FUNCTION "FC2027_ZC_FF_SEC" : Void
TITLE = FC2027_FF_SEC
{ S7_Optimized_Access := 'TRUE' }
AUTHOR : ABH
FAMILY : ZeusControl
VERSION : 1.0
//Funcion para gestion de Flip Flop secuencial.
   VAR_INPUT
      Pulso1Seg : Bool;   // Pulso de 1 segundo
   END_VAR

   VAR_TEMP
      for_i : Int;
      t_Flip_1 : Int;
      t_Flip_2 : Int;
      t_Flip_3 : Int;
      t_Flip_4 : Int;
      t_Flip_5 : Int;
      t_Flip_6 : Int;
      t_Flip_7 : Int;
      t_Flip_8 : Int;
      t_Flip_9 : Int;
      t_Flip_10 : Int;
   END_VAR


BEGIN
	(*
	ZEUS CONTROL, S.A.
	(c)Copyright (2023) All Rights Reserved
	--------------------------------------------------------------------------------------

	Software:       TIA Portal 16
	Restricciones:  PLC serie 1200/1500

	Nombre:         DISPOSITIVO FLIP FLOP SECUENCIAL
	Descripcion:    Modelo de dispositivo Flip Flop Secuencial

	Dependencias:
	    FC:         -
	    FB:         -
	    UDT:        ZC_DISP_FF_SEC
	    DB:         DB2027_DISP_FF_SEC

	Change log:

	    Version     Fecha       Tecnico a cargo     Descripcion

	    01.00.00    23.06.2022  (ABH)               Primera version
	    01.00.01    15.07.2022  (HCR)               Se aumenta la gestion de flips de 6 a 10.
	    01.00.02    28.11.2023  (ABH)               Se añade condicion de activacion del Flip Flop a que algun SP sea mayor que 0.
	    01.00.03    15.10.2025  (ABH)               Se añade orden pausa para dejar de contar.

	//=====================================================================================
	*)



	FOR #for_i := 1 TO "N_MAX_DISP_FF_SEC" DO


	    IF "DB2027_FF_SEC".FF_SEC[#for_i].Orden_Activar AND
	        ("DB2027_FF_SEC".FF_SEC[#for_i].Config_SetPointTiempoFlip1 > 0
	        OR"DB2027_FF_SEC".FF_SEC[#for_i].Config_SetPointTiempoFlip2 > 0
	        OR"DB2027_FF_SEC".FF_SEC[#for_i].Config_SetPointTiempoFlip3 > 0
	        OR"DB2027_FF_SEC".FF_SEC[#for_i].Config_SetPointTiempoFlip4 > 0
	        OR"DB2027_FF_SEC".FF_SEC[#for_i].Config_SetPointTiempoFlip5 > 0
	        OR"DB2027_FF_SEC".FF_SEC[#for_i].Config_SetPointTiempoFlip6 > 0
	        OR"DB2027_FF_SEC".FF_SEC[#for_i].Config_SetPointTiempoFlip7 > 0
	        OR"DB2027_FF_SEC".FF_SEC[#for_i].Config_SetPointTiempoFlip8 > 0
	        OR"DB2027_FF_SEC".FF_SEC[#for_i].Config_SetPointTiempoFlip9 > 0
	        OR"DB2027_FF_SEC".FF_SEC[#for_i].Config_SetPointTiempoFlip10 > 0
	        OR"DB2027_FF_SEC".FF_SEC[#for_i].Config_SetPointTiempoFlop > 0)
	    THEN



	        REGION ARRANQUE_ACTIVACION_FLOP

	            //  EN EL ARRANQUE SE ACTIVA FLOP
	            IF "DB2027_FF_SEC".FF_SEC[#for_i].Aux_Flanco = FALSE THEN
	                "DB2027_FF_SEC".FF_SEC[#for_i].Aux_FlopActivo := TRUE;
	                "DB2027_FF_SEC".FF_SEC[#for_i].Aux_FlipActivo := FALSE;
	                "DB2027_FF_SEC".FF_SEC[#for_i].Aux_Flanco := TRUE;
	            END_IF;

	        END_REGION


	        REGION CALCULO_TIEMPOS_FLIP

	            //  CALCULO DE ACTIVACIONES SECUENCIALES
	            #t_Flip_1 := "DB2027_FF_SEC".FF_SEC[#for_i].Config_SetPointTiempoFlip1;
	            #t_Flip_2 := #t_Flip_1 + "DB2027_FF_SEC".FF_SEC[#for_i].Config_SetPointTiempoFlip2;
	            #t_Flip_3 := #t_Flip_2 + "DB2027_FF_SEC".FF_SEC[#for_i].Config_SetPointTiempoFlip3;
	            #t_Flip_4 := #t_Flip_3 + "DB2027_FF_SEC".FF_SEC[#for_i].Config_SetPointTiempoFlip4;
	            #t_Flip_5 := #t_Flip_4 + "DB2027_FF_SEC".FF_SEC[#for_i].Config_SetPointTiempoFlip5;
	            #t_Flip_6 := #t_Flip_5 + "DB2027_FF_SEC".FF_SEC[#for_i].Config_SetPointTiempoFlip6;
	            #t_Flip_7 := #t_Flip_6 + "DB2027_FF_SEC".FF_SEC[#for_i].Config_SetPointTiempoFlip7;
	            #t_Flip_8 := #t_Flip_7 + "DB2027_FF_SEC".FF_SEC[#for_i].Config_SetPointTiempoFlip8;
	            #t_Flip_9 := #t_Flip_8 + "DB2027_FF_SEC".FF_SEC[#for_i].Config_SetPointTiempoFlip9;
	            #t_Flip_10 := #t_Flip_9 + "DB2027_FF_SEC".FF_SEC[#for_i].Config_SetPointTiempoFlip10;

	            //  CALCULO DE TIEMPO FLIP TOTAL
	            "DB2027_FF_SEC".FF_SEC[#for_i].Aux_TiempoFlipTotal :=
	            "DB2027_FF_SEC".FF_SEC[#for_i].Config_SetPointTiempoFlip1 +
	            "DB2027_FF_SEC".FF_SEC[#for_i].Config_SetPointTiempoFlip2 +
	            "DB2027_FF_SEC".FF_SEC[#for_i].Config_SetPointTiempoFlip3 +
	            "DB2027_FF_SEC".FF_SEC[#for_i].Config_SetPointTiempoFlip4 +
	            "DB2027_FF_SEC".FF_SEC[#for_i].Config_SetPointTiempoFlip5 +
	            "DB2027_FF_SEC".FF_SEC[#for_i].Config_SetPointTiempoFlip6 +
	            "DB2027_FF_SEC".FF_SEC[#for_i].Config_SetPointTiempoFlip7 +
	            "DB2027_FF_SEC".FF_SEC[#for_i].Config_SetPointTiempoFlip8 +
	            "DB2027_FF_SEC".FF_SEC[#for_i].Config_SetPointTiempoFlip9 +
	            "DB2027_FF_SEC".FF_SEC[#for_i].Config_SetPointTiempoFlip10;

	        END_REGION


	        REGION ACTIVACION_FLIP_FLOP

	            //  GESTION FLIP
	            IF "DB2027_FF_SEC".FF_SEC[#for_i].Aux_TiempoFlip >= "DB2027_FF_SEC".FF_SEC[#for_i].Aux_TiempoFlipTotal THEN

	                "DB2027_FF_SEC".FF_SEC[#for_i].Aux_TiempoFlip := 0;
	                "DB2027_FF_SEC".FF_SEC[#for_i].Aux_FlipActivo := FALSE;
	                "DB2027_FF_SEC".FF_SEC[#for_i].Aux_FlopActivo := TRUE;

	            END_IF;

	            //  GESTION FLOP
	            IF "DB2027_FF_SEC".FF_SEC[#for_i].Aux_TiempoFlop >= "DB2027_FF_SEC".FF_SEC[#for_i].Config_SetPointTiempoFlop THEN

	                "DB2027_FF_SEC".FF_SEC[#for_i].Aux_TiempoFlop := 0;
	                "DB2027_FF_SEC".FF_SEC[#for_i].Aux_FlipActivo := TRUE;
	                "DB2027_FF_SEC".FF_SEC[#for_i].Aux_FlopActivo := FALSE;

	            END_IF;

	        END_REGION


	        REGION CONTAJE_TIEMPOS_FLIP_FLOP

	            IF #Pulso1Seg AND NOT "DB2027_FF_SEC".FF_SEC[#for_i].Orden_Pausa THEN

	                //  CUENTA FLIP
	                IF "DB2027_FF_SEC".FF_SEC[#for_i].Aux_FlipActivo THEN
	                    "DB2027_FF_SEC".FF_SEC[#for_i].Aux_TiempoFlip += + 1;
	                END_IF;

	                //  CUENTA FLOP
	                IF "DB2027_FF_SEC".FF_SEC[#for_i].Aux_FlopActivo THEN
	                    "DB2027_FF_SEC".FF_SEC[#for_i].Aux_TiempoFlop += + 1;
	                END_IF;

	            END_IF;

	        END_REGION


	        REGION ACTIVACION_SALIDAS

	            // GESTION SALIDAS FLOP
	            IF "DB2027_FF_SEC".FF_SEC[#for_i].Aux_FlopActivo THEN

	                "DB2027_FF_SEC".FF_SEC[#for_i].Estado_SalidaFlop := TRUE;

	                "DB2027_FF_SEC".FF_SEC[#for_i].Estado_SalidaFlip1 :=
	                "DB2027_FF_SEC".FF_SEC[#for_i].Estado_SalidaFlip2 :=
	                "DB2027_FF_SEC".FF_SEC[#for_i].Estado_SalidaFlip3 :=
	                "DB2027_FF_SEC".FF_SEC[#for_i].Estado_SalidaFlip4 :=
	                "DB2027_FF_SEC".FF_SEC[#for_i].Estado_SalidaFlip5 :=
	                "DB2027_FF_SEC".FF_SEC[#for_i].Estado_SalidaFlip6 :=
	                "DB2027_FF_SEC".FF_SEC[#for_i].Estado_SalidaFlip7 :=
	                "DB2027_FF_SEC".FF_SEC[#for_i].Estado_SalidaFlip8 :=
	                "DB2027_FF_SEC".FF_SEC[#for_i].Estado_SalidaFlip9 :=
	                "DB2027_FF_SEC".FF_SEC[#for_i].Estado_SalidaFlip10 := FALSE;
	            END_IF;

	            // GESTION SALIDAS FLIP
	            IF "DB2027_FF_SEC".FF_SEC[#for_i].Aux_FlipActivo THEN

	                //  ACTIVACION FLIP 1
	                IF "DB2027_FF_SEC".FF_SEC[#for_i].Aux_TiempoFlip < #t_Flip_1 AND "DB2027_FF_SEC".FF_SEC[#for_i].Config_SetPointTiempoFlip1 <> 0 THEN
	                    "DB2027_FF_SEC".FF_SEC[#for_i].Estado_SalidaFlip1 := TRUE;
	                ELSE
	                    "DB2027_FF_SEC".FF_SEC[#for_i].Estado_SalidaFlip1 := FALSE;
	                END_IF;

	                //  ACTIVACION FLIP 2
	                IF "DB2027_FF_SEC".FF_SEC[#for_i].Aux_TiempoFlip >= #t_Flip_1 AND "DB2027_FF_SEC".FF_SEC[#for_i].Aux_TiempoFlip < #t_Flip_2 AND "DB2027_FF_SEC".FF_SEC[#for_i].Config_SetPointTiempoFlip2 <> 0 THEN
	                    "DB2027_FF_SEC".FF_SEC[#for_i].Estado_SalidaFlip2 := TRUE;
	                ELSE
	                    "DB2027_FF_SEC".FF_SEC[#for_i].Estado_SalidaFlip2 := FALSE;
	                END_IF;

	                //  ACTIVACION FLIP 3
	                IF "DB2027_FF_SEC".FF_SEC[#for_i].Aux_TiempoFlip >= #t_Flip_2 AND "DB2027_FF_SEC".FF_SEC[#for_i].Aux_TiempoFlip < #t_Flip_3 AND "DB2027_FF_SEC".FF_SEC[#for_i].Config_SetPointTiempoFlip3 <> 0 THEN
	                    "DB2027_FF_SEC".FF_SEC[#for_i].Estado_SalidaFlip3 := TRUE;
	                ELSE
	                    "DB2027_FF_SEC".FF_SEC[#for_i].Estado_SalidaFlip3 := FALSE;
	                END_IF;

	                //  ACTIVACION FLIP 4
	                IF "DB2027_FF_SEC".FF_SEC[#for_i].Aux_TiempoFlip >= #t_Flip_3 AND "DB2027_FF_SEC".FF_SEC[#for_i].Aux_TiempoFlip < #t_Flip_4 AND "DB2027_FF_SEC".FF_SEC[#for_i].Config_SetPointTiempoFlip4 <> 0 THEN
	                    "DB2027_FF_SEC".FF_SEC[#for_i].Estado_SalidaFlip4 := TRUE;
	                ELSE
	                    "DB2027_FF_SEC".FF_SEC[#for_i].Estado_SalidaFlip4 := FALSE;
	                END_IF;

	                //  ACTIVACION FLIP 5
	                IF "DB2027_FF_SEC".FF_SEC[#for_i].Aux_TiempoFlip >= #t_Flip_4 AND "DB2027_FF_SEC".FF_SEC[#for_i].Aux_TiempoFlip < #t_Flip_5 AND "DB2027_FF_SEC".FF_SEC[#for_i].Config_SetPointTiempoFlip5 <> 0 THEN
	                    "DB2027_FF_SEC".FF_SEC[#for_i].Estado_SalidaFlip5 := TRUE;
	                ELSE
	                    "DB2027_FF_SEC".FF_SEC[#for_i].Estado_SalidaFlip5 := FALSE;
	                END_IF;

	                //  ACTIVACION FLIP 6
	                IF "DB2027_FF_SEC".FF_SEC[#for_i].Aux_TiempoFlip >= #t_Flip_5 AND "DB2027_FF_SEC".FF_SEC[#for_i].Aux_TiempoFlip < #t_Flip_6 AND "DB2027_FF_SEC".FF_SEC[#for_i].Config_SetPointTiempoFlip6 <> 0 THEN
	                    "DB2027_FF_SEC".FF_SEC[#for_i].Estado_SalidaFlip6 := TRUE;
	                ELSE
	                    "DB2027_FF_SEC".FF_SEC[#for_i].Estado_SalidaFlip6 := FALSE;
	                END_IF;

	                //  ACTIVACION FLIP 7
	                IF "DB2027_FF_SEC".FF_SEC[#for_i].Aux_TiempoFlip >= #t_Flip_6 AND "DB2027_FF_SEC".FF_SEC[#for_i].Aux_TiempoFlip < #t_Flip_7 AND "DB2027_FF_SEC".FF_SEC[#for_i].Config_SetPointTiempoFlip7 <> 0 THEN
	                    "DB2027_FF_SEC".FF_SEC[#for_i].Estado_SalidaFlip7 := TRUE;
	                ELSE
	                    "DB2027_FF_SEC".FF_SEC[#for_i].Estado_SalidaFlip7 := FALSE;
	                END_IF;

	                //  ACTIVACION FLIP 8
	                IF "DB2027_FF_SEC".FF_SEC[#for_i].Aux_TiempoFlip >= #t_Flip_7 AND "DB2027_FF_SEC".FF_SEC[#for_i].Aux_TiempoFlip < #t_Flip_8 AND "DB2027_FF_SEC".FF_SEC[#for_i].Config_SetPointTiempoFlip8 <> 0 THEN
	                    "DB2027_FF_SEC".FF_SEC[#for_i].Estado_SalidaFlip8 := TRUE;
	                ELSE
	                    "DB2027_FF_SEC".FF_SEC[#for_i].Estado_SalidaFlip8 := FALSE;
	                END_IF;

	                //  ACTIVACION FLIP 9
	                IF "DB2027_FF_SEC".FF_SEC[#for_i].Aux_TiempoFlip >= #t_Flip_8 AND "DB2027_FF_SEC".FF_SEC[#for_i].Aux_TiempoFlip < #t_Flip_9 AND "DB2027_FF_SEC".FF_SEC[#for_i].Config_SetPointTiempoFlip9 <> 0 THEN
	                    "DB2027_FF_SEC".FF_SEC[#for_i].Estado_SalidaFlip9 := TRUE;
	                ELSE
	                    "DB2027_FF_SEC".FF_SEC[#for_i].Estado_SalidaFlip9 := FALSE;
	                END_IF;

	                //  ACTIVACION FLIP 10
	                IF "DB2027_FF_SEC".FF_SEC[#for_i].Aux_TiempoFlip >= #t_Flip_9 AND "DB2027_FF_SEC".FF_SEC[#for_i].Aux_TiempoFlip < #t_Flip_10 AND "DB2027_FF_SEC".FF_SEC[#for_i].Config_SetPointTiempoFlip10 <> 0 THEN
	                    "DB2027_FF_SEC".FF_SEC[#for_i].Estado_SalidaFlip10 := TRUE;
	                ELSE
	                    "DB2027_FF_SEC".FF_SEC[#for_i].Estado_SalidaFlip10 := FALSE;
	                END_IF;


	                "DB2027_FF_SEC".FF_SEC[#for_i].Estado_SalidaFlop := FALSE;
	            END_IF;

	        END_REGION

	    ELSE

	        "DB2027_FF_SEC".FF_SEC[#for_i].Aux_TiempoFlip :=
	        "DB2027_FF_SEC".FF_SEC[#for_i].Aux_TiempoFlop := 0;
	        "DB2027_FF_SEC".FF_SEC[#for_i].Estado_SalidaFlop :=
	        "DB2027_FF_SEC".FF_SEC[#for_i].Estado_SalidaFlip1 :=
	        "DB2027_FF_SEC".FF_SEC[#for_i].Estado_SalidaFlip2 :=
	        "DB2027_FF_SEC".FF_SEC[#for_i].Estado_SalidaFlip3 :=
	        "DB2027_FF_SEC".FF_SEC[#for_i].Estado_SalidaFlip4 :=
	        "DB2027_FF_SEC".FF_SEC[#for_i].Estado_SalidaFlip5 :=
	        "DB2027_FF_SEC".FF_SEC[#for_i].Estado_SalidaFlip6 :=
	        "DB2027_FF_SEC".FF_SEC[#for_i].Estado_SalidaFlip7 :=
	        "DB2027_FF_SEC".FF_SEC[#for_i].Estado_SalidaFlip8 :=
	        "DB2027_FF_SEC".FF_SEC[#for_i].Estado_SalidaFlip9 :=
	        "DB2027_FF_SEC".FF_SEC[#for_i].Estado_SalidaFlip10 := FALSE;

	        "DB2027_FF_SEC".FF_SEC[#for_i].Aux_FlipActivo := FALSE;
	        "DB2027_FF_SEC".FF_SEC[#for_i].Aux_FlopActivo := TRUE;

	        "DB2027_FF_SEC".FF_SEC[#for_i].Aux_Flanco := FALSE;

	    END_IF;

	END_FOR;
END_FUNCTION

